Fanuc KAREL source: kt00236.KL

-- PROVISIONAL review KL for V770-1; original PC SHA256 053529e2f2428222a74278b2e63a95873768a33d078ad5aa941414f56dbf5741
-- Incomplete behavior may be omitted. Consult companion uncertainty JSON. Do not deploy.
PROGRAM KT00236
%NOLOCKGROUP
VAR
  I1 : INTEGER
  I2 : INTEGER
  OUT : INTEGER
BEGIN
  -- UNRESOLVED_PC offsets 5-16; opcodes 2E,23
  -- UNRESOLVED_PC offsets 21-32; opcodes 2E,23
  -- UNRESOLVED_PC offsets 37-48; opcodes 2E,23
  -- UNRESOLVED_PC offsets 53-64; opcodes 2E,23
  -- UNRESOLVED_PC offsets 69-88; opcodes 21,21,47,23
  -- UNRESOLVED_PC offsets 93-97; opcodes 7F
END KT00236
